FUNCTION_BLOCK ClamperFilterSide EXTENDS RunUnitSlave
VAR_INPUT
END_VAR
VAR_OUTPUT
END_VAR
VAR
END_VAR

END_FUNCTION_BLOCK

(* stored: Version 1.1.0.1, ProductVersion 3.1.4024.0
   POU ClamperFilterSide: Id {4cfbb8e7-dd19-45d2-8e96-6129406da078}, SpecialFunc None *)
